% RSLogix 500 project PLC TASK - CONVEYOR WITH JAM DETECTION_BAK000.RSS, saved by version 8.30.00.16 %
PROJECT "UNTITLED"    % processor: Bul.1763 MicroLogix 1100 Series B %

PROGRAM FILES
  LAD 2 "MAIN"  3 rungs
  LAD 3 "DIGITAL IO"  12 rungs
  LAD 4 "CONTROLS"  6 rungs

DATA FILES
  O0 OUTPUT  5 elements
  I1 INPUT  7 elements
  S2 STATUS  66 elements
  B3 BINARY  1 elements
  T4 TIMER  1 elements
  C5 COUNTER  1 elements
  R6 CONTROL  1 elements
  N7 INTEGER  1 elements
  F8 FLOAT  1 elements

LADDER 2 "MAIN"
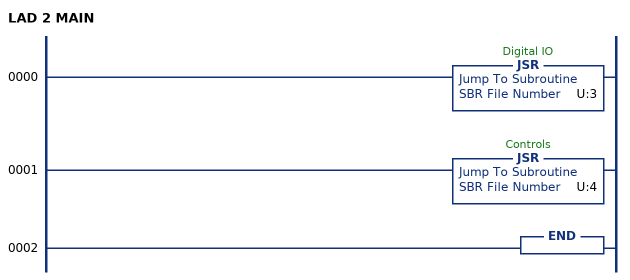
% Rung: 0 %  % edit flag set %
SOR JSR U:3 EOR
%   U:3  "Digital IO" %
% Rung: 1 %  % edit flag set %
SOR JSR U:4 EOR
%   U:4  "Controls" %
% Rung: 2 %
SOR END EOR

LADDER 3 "DIGITAL IO"
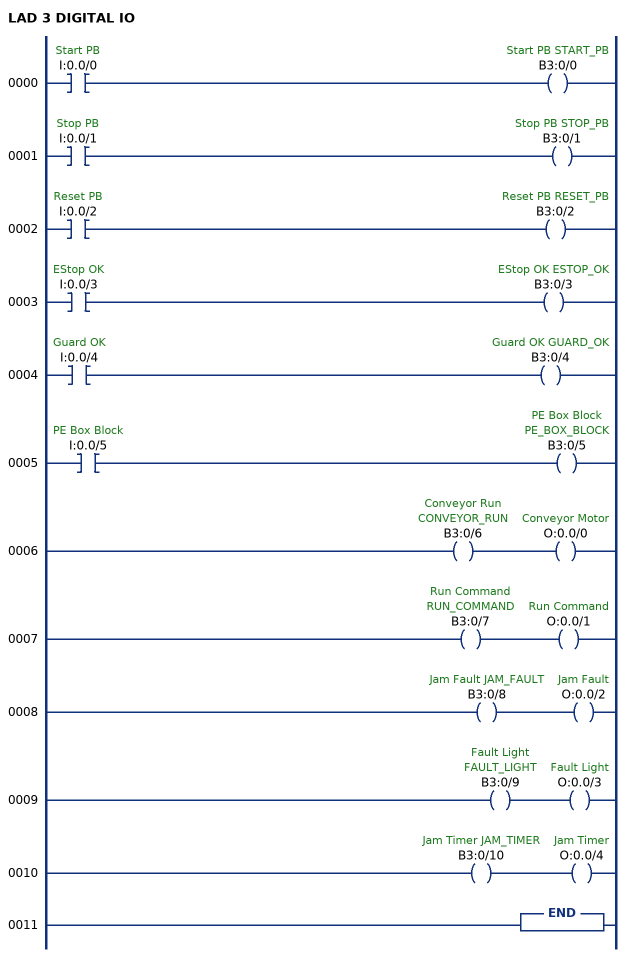
% Rung: 0 %  % edit flag set %
SOR XIC I:0.0/0 OTE B3:0/0 EOR
%   I:0.0/0  "Start PB" %
%   B3:0/0  START_PB  "Start PB" %
% Rung: 1 %  % edit flag set %
SOR XIC I:0.0/1 OTE B3:0/1 EOR
%   I:0.0/1  "Stop PB" %
%   B3:0/1  STOP_PB  "Stop PB" %
% Rung: 2 %  % edit flag set %
SOR XIC I:0.0/2 OTE B3:0/2 EOR
%   I:0.0/2  "Reset PB" %
%   B3:0/2  RESET_PB  "Reset PB" %
% Rung: 3 %  % edit flag set %
SOR XIC I:0.0/3 OTE B3:0/3 EOR
%   I:0.0/3  "EStop OK" %
%   B3:0/3  ESTOP_OK  "EStop OK" %
% Rung: 4 %  % edit flag set %
SOR XIC I:0.0/4 OTE B3:0/4 EOR
%   I:0.0/4  "Guard OK" %
%   B3:0/4  GUARD_OK  "Guard OK" %
% Rung: 5 %  % edit flag set %
SOR XIC I:0.0/5 OTE B3:0/5 EOR
%   I:0.0/5  "PE Box Block" %
%   B3:0/5  PE_BOX_BLOCK  "PE Box Block" %
% Rung: 6 %  % edit flag set %
SOR OTE B3:0/6 OTE O:0.0/0 EOR
%   B3:0/6  CONVEYOR_RUN  "Conveyor Run" %
%   O:0.0/0  "Conveyor Motor" %
% Rung: 7 %  % edit flag set %
SOR OTE B3:0/7 OTE O:0.0/1 EOR
%   B3:0/7  RUN_COMMAND  "Run Command" %
%   O:0.0/1  "Run Command" %
% Rung: 8 %  % edit flag set %
SOR OTE B3:0/8 OTE O:0.0/2 EOR
%   B3:0/8  JAM_FAULT  "Jam Fault" %
%   O:0.0/2  "Jam Fault" %
% Rung: 9 %  % edit flag set %
SOR OTE B3:0/9 OTE O:0.0/3 EOR
%   B3:0/9  FAULT_LIGHT  "Fault Light" %
%   O:0.0/3  "Fault Light" %
% Rung: 10 %  % edit flag set %
SOR OTE B3:0/10 OTE O:0.0/4 EOR
%   B3:0/10  JAM_TIMER  "Jam Timer" %
%   O:0.0/4  "Jam Timer" %
% Rung: 11 %
SOR END EOR

LADDER 4 "CONTROLS"
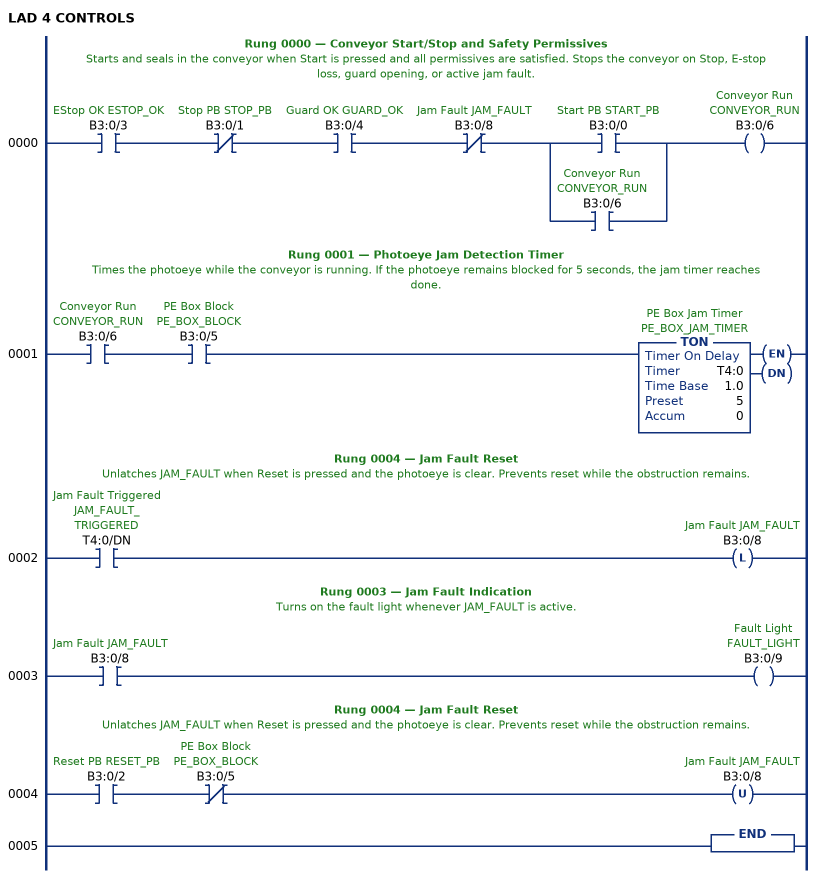
% Rung: 0 %  % edit flag set %
% TITLE: Rung 0000 — Conveyor Start/Stop and Safety Permissives %
% Starts and seals in the conveyor when Start is pressed and all permissives are satisfied. Stops the conveyor on Stop, E-stop loss, guard opening, or active jam fault. %
SOR XIC B3:0/3 XIO B3:0/1 XIC B3:0/4 XIO B3:0/8 BST XIC B3:0/0 NXB XIC B3:0/6 BND OTE B3:0/6 EOR
%   B3:0/3  ESTOP_OK  "EStop OK" %
%   B3:0/1  STOP_PB  "Stop PB" %
%   B3:0/4  GUARD_OK  "Guard OK" %
%   B3:0/8  JAM_FAULT  "Jam Fault" %
%   B3:0/0  START_PB  "Start PB" %
%   B3:0/6  CONVEYOR_RUN  "Conveyor Run" %
% Rung: 1 %  % edit flag set %
% TITLE: Rung 0001 — Photoeye Jam Detection Timer %
% Times the photoeye while the conveyor is running. If the photoeye remains blocked for 5 seconds, the jam timer reaches done. %
SOR XIC B3:0/6 XIC B3:0/5 TON T4:0 1.0 5 0 EOR
%   B3:0/6  CONVEYOR_RUN  "Conveyor Run" %
%   B3:0/5  PE_BOX_BLOCK  "PE Box Block" %
%   T4:0  PE_BOX_JAM_TIMER  "PE Box Jam Timer" %
% Rung: 2 %  % edit flag set %
% TITLE: Rung 0004 — Jam Fault Reset %
% Unlatches JAM_FAULT when Reset is pressed and the photoeye is clear. Prevents reset while the obstruction remains. %
SOR XIC T4:0/DN OTL B3:0/8 EOR
%   T4:0/DN  JAM_FAULT_TRIGGERED  "Jam Fault Triggered" %
%   B3:0/8  JAM_FAULT  "Jam Fault" %
% Rung: 3 %  % edit flag set %
% TITLE: Rung 0003 — Jam Fault Indication %
% Turns on the fault light whenever JAM_FAULT is active. %
SOR XIC B3:0/8 OTE B3:0/9 EOR
%   B3:0/8  JAM_FAULT  "Jam Fault" %
%   B3:0/9  FAULT_LIGHT  "Fault Light" %
% Rung: 4 %  % edit flag set %
% TITLE: Rung 0004 — Jam Fault Reset %
% Unlatches JAM_FAULT when Reset is pressed and the photoeye is clear. Prevents reset while the obstruction remains. %
SOR XIC B3:0/2 XIO B3:0/5 OTU B3:0/8 EOR
%   B3:0/2  RESET_PB  "Reset PB" %
%   B3:0/5  PE_BOX_BLOCK  "PE Box Block" %
%   B3:0/8  JAM_FAULT  "Jam Fault" %
% Rung: 5 %
SOR END EOR
